(****************************************************************************************)
(*							Beckhoff Automation Poland									*)
(*									F_1stByteW	v1.0									*)
(*									15.02.2010											*)
(*		Funkcja wyciagajaca mniej znaczacy BYTE ze zmiennej typu WORD					*)
(*							 wyjscie typu WORD											*)
(*______________________________________________________________________________________*)
FUNCTION F_1stByteW : WORD
VAR_INPUT
	wIn:	WORD;
END_VAR

F_1stByteW := wIn AND 16#FF;

END_FUNCTION

(* stored: Version 1.1.0.1, ProductVersion 3.1.4026.13, FileIdentifier 5269eff6b6f053316505e33648e8511c2dd7467a, FileSignature 3c7fc476c0f8c13b680f4f2a6acc69f727c14453591f27a5cd525b77b304c4e3105df0e65055cfa61826486e8c0b4a20a742fc23675bc818e8bb732a5b101a6c367f35f43220d8ab6652d2b488985205a8d6511fd43f0d82b813e2ae0ac261eeb74c6ea8551bc8d5700641aec9e301d3e8558fca589f7fb29869613f7a4fd26c3305e10e7e54a1f9b549afc627b03ce0b50b3e3d173163812bdc7c7701a9329d68ec6f52fb9b8d7c3d3582032856f87f742ad4ec3c69b816df2b48177482d4769fd1eec265775e8e99e4e70ddf17de93ee1f68114d3eb7d0dfc0540818439f75dea5d3a15e20f618523046ac8407c192bda22715c773bd468c07bbb8be599786
   POU F_1stByteW: Id {2548d8cf-d639-4a8e-b341-312f9939f085}, SpecialFunc None *)
